TYPE ConditionConfig :
STRUCT
	symbol		: __SYSTEM.AnyType;
	
	index		: UINT;
END_STRUCT
END_TYPE

(* stored: Version 1.1.0.1, ProductVersion 3.1.4024.11
   DUT ConditionConfig: Id {eb28fe82-d717-4247-8f44-545d36f05065} *)
